// Mitsubishi GX Works2 project: 최예현   PLC: Q02/Q02H

PROGRAM MAIN
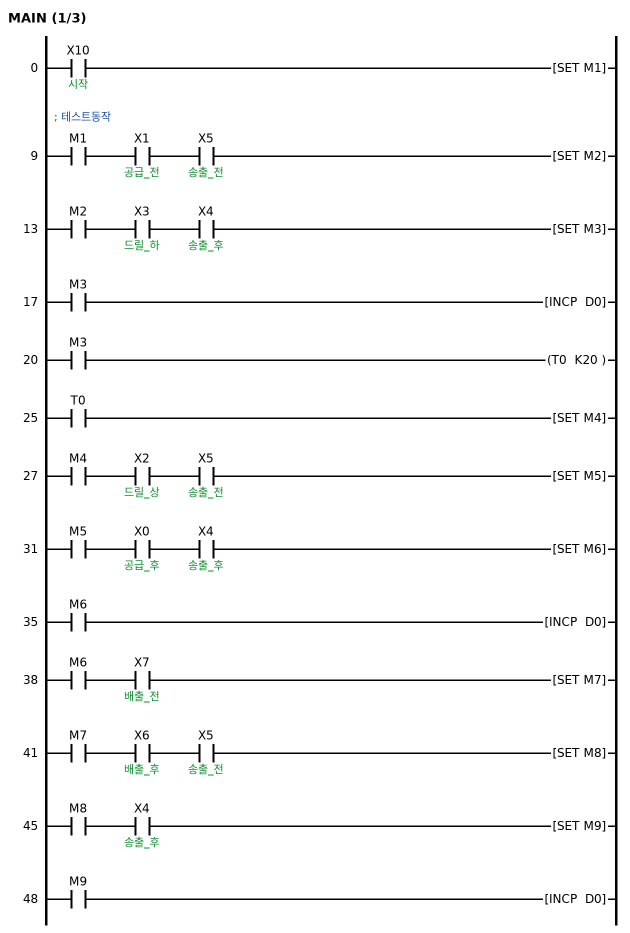
0     LD      X10  ; 시작
      SET     M1
; 테스트동작
9     LD      M1
      AND     X1  ; 공급_전
      AND     X5  ; 송출_전
      SET     M2
13    LD      M2
      AND     X3  ; 드릴_하
      AND     X4  ; 송출_후
      SET     M3
17    LD      M3
      INCP    D0
20    LD      M3
      OUT     T0 K20
25    LD      T0
      SET     M4
27    LD      M4
      AND     X2  ; 드릴_상
      AND     X5  ; 송출_전
      SET     M5
31    LD      M5
      AND     X0  ; 공급_후
      AND     X4  ; 송출_후
      SET     M6
35    LD      M6
      INCP    D0
38    LD      M6
      AND     X7  ; 배출_전
      SET     M7
41    LD      M7
      AND     X6  ; 배출_후
      AND     X5  ; 송출_전
      SET     M8
45    LD      M8
      AND     X4  ; 송출_후
      SET     M9
48    LD      M9
      INCP    D0
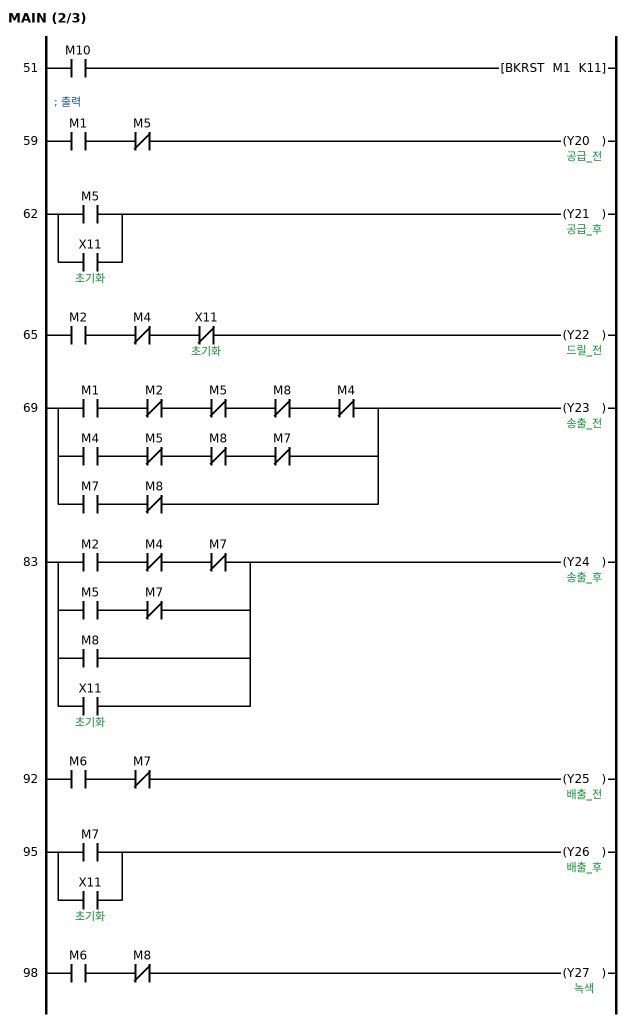
51    LD      M10
      BKRST   M1 K11
; 출력
59    LD      M1
      ANI     M5
      OUT     Y20  ; 공급_전
62    LD      M5
      OR      X11  ; 초기화
      OUT     Y21  ; 공급_후
65    LD      M2
      ANI     M4
      ANI     X11  ; 초기화
      OUT     Y22  ; 드릴_전
69    LD      M1
      ANI     M2
      ANI     M5
      ANI     M8
      ANI     M4
      LD      M4
      ANI     M5
      ANI     M8
      ANI     M7
      ORB
      LD      M7
      ANI     M8
      ORB
      OUT     Y23  ; 송출_전
83    LD      M2
      ANI     M4
      ANI     M7
      LD      M5
      ANI     M7
      ORB
      OR      M8
      OR      X11  ; 초기화
      OUT     Y24  ; 송출_후
92    LD      M6
      ANI     M7
      OUT     Y25  ; 배출_전
95    LD      M7
      OR      X11  ; 초기화
      OUT     Y26  ; 배출_후
98    LD      M6
      ANI     M8
      OUT     Y27  ; 녹색
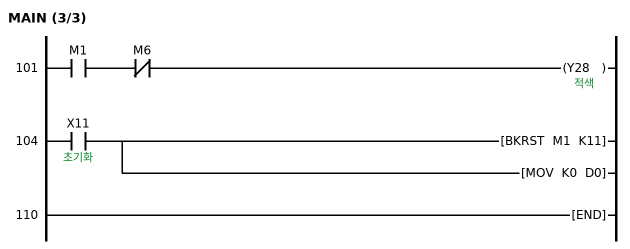
101   LD      M1
      ANI     M6
      OUT     Y28  ; 적색
104   LD      X11  ; 초기화
      BKRST   M1 K11
      MOV     K0 D0
110   END
END_PROGRAM

PROGRAM HMI
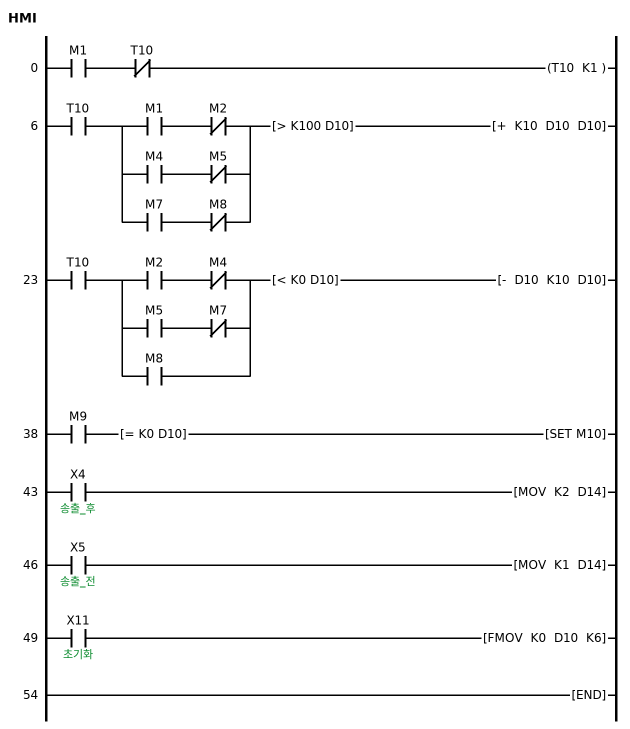
0     LD      M1
      ANI     T10
      OUT     T10 K1
6     LD      T10
      LD      M1
      ANI     M2
      LD      M4
      ANI     M5
      ORB
      LD      M7
      ANI     M8
      ORB
      ANB
      AND>    K100 D10
      +       K10 D10 D10
23    LD      T10
      LD      M2
      ANI     M4
      LD      M5
      ANI     M7
      ORB
      OR      M8
      ANB
      AND<    K0 D10
      -       D10 K10 D10
38    LD      M9
      AND=    K0 D10
      SET     M10
43    LD      X4  ; 송출_후
      MOV     K2 D14
46    LD      X5  ; 송출_전
      MOV     K1 D14
49    LD      X11  ; 초기화
      FMOV    K0 D10 K6
54    END
END_PROGRAM
